{attribute 'linkalways'} 
{attribute 'no_explicit_call' := 'This FB is a CLASS and must be accessed using methods or properties'}
{attribute 'enable_dynamic_creation'}
FUNCTION_BLOCK _TIMESTRUCT EXTENDS StructuredDatatypeBase
VAR
	localData : TIMESTRUCT;
	activeData : REFERENCE TO TIMESTRUCT REF= localData;
	_wYear : _WORD(localData.wYear);
	_wMonth : _WORD(localData.wMonth);
END_VAR

PROPERTY PUBLIC Address : PVOID
GET
Address := ADR(activeData);
END_GET
END_PROPERTY

METHOD PUBLIC ClearReference
VAR_INPUT
END_VAR
activeData REF= localData;
END_METHOD

METHOD PUBLIC Clone : I_Datatype
VAR
    pClone : POINTER TO _TIMESTRUCT;
END_VAR
pClone := __NEW(_TIMESTRUCT());
pClone^.Value := Value;
Clone := pClone^;
END_METHOD

PROPERTY PUBLIC Identifier : T_MAXSTRING
GET
Identifier := 'TIMESTRUCT';
END_GET
END_PROPERTY

METHOD PROTECTED InitializeMembers
VAR_INPUT
	members : REFERENCE TO MembersHost;
END_VAR
_wYear.MakeReferenceTo(activeData.wYear);
members.AddMember('wYear',_wYear);

_wMonth.MakeReferenceTo(activeData.wMonth);
members.AddMember('wMonth',_wMonth);
END_METHOD

METHOD PUBLIC MakeReferenceTo
VAR_INPUT
	ReferenceTarget : TIMESTRUCT;
END_VAR
activeData REF= ReferenceTarget;
END_METHOD

PROPERTY PUBLIC Size : UDINT
GET
Size := SIZEOF(activeData);
END_GET
END_PROPERTY

METHOD TryMakeReferenceTo : BOOL
VAR_INPUT
	Target : I_Datatype;
END_VAR
VAR
	pTargetData : POINTER TO TIMESTRUCT;
END_VAR
IF NOT (Target.IecType = IecType) THEN
	RETURN;
END_IF

pTargetData := Target.Address;
activeData REF= pTargetData^;
TryMakeReferenceTo := TRUE;
END_METHOD

PROPERTY PUBLIC Value : TIMESTRUCT
GET
Value := activeData;
END_GET
SET
activeData := Value;
END_SET
END_PROPERTY

PROPERTY PUBLIC wMonth : Reference to _WORD
GET
wMonth := _wMonth;
END_GET
END_PROPERTY

PROPERTY PUBLIC wYear : Reference to _WORD
GET
wYear := _wYear;
END_GET
END_PROPERTY

END_FUNCTION_BLOCK

(* stored: Version 1.1.0.1, ProductVersion 3.1.4024.12
   POU _TIMESTRUCT: Id {82e9ef09-f63f-071f-12cd-f370d2802325}, SpecialFunc None
   Folder Protected: Id {9fdedf6e-4ca0-00e0-0273-13cb491dabf3}
   Property Address: Id {b5129746-2857-0022-1d98-5cd0054c1e32}
   Get Get: Id {b9ad7187-0100-02be-2dd1-43dd70cfdd46}
   Method ClearReference: Id {16c22b7d-2069-0e94-0823-7f69befe1715}
   Method Clone: Id {f9cc5498-2141-4519-8b72-11d757b9f1bd}
   Property Identifier: Id {11804f6c-c92e-0f5b-382d-3367d277dbcc}
   Get Get: Id {7977c071-5d37-04dd-33f0-5d682f8e3abf}
   Method InitializeMembers: Id {59fd7717-5550-0f25-158c-9c1e87cde269}
   Method MakeReferenceTo: Id {7e8e9cd2-b76b-014b-0b95-9790b062a9ee}
   Property Size: Id {3db85a58-3871-08be-0a1b-c8cbab28906e}
   Get Get: Id {c45ad51d-3dc4-00ea-11f7-a16d1bad1963}
   Method TryMakeReferenceTo: Id {8b5d5a6b-3b1b-05bb-2e0f-edb7929e5540}
   Property Value: Id {b58f9a32-1b3b-0a05-0577-0e7b74707ce6}
   Get Get: Id {d1a2ef74-1fb0-0703-20c2-eb9eec1cc598}
   Set Set: Id {4bd1c6bf-61b3-0a38-37ec-840667c35baf}
   Property wMonth: Id {54bb8911-1454-0b68-0e6e-66985ac5d437}
   Get Get: Id {8a1a1f3d-9a7a-02bf-2086-eb0b47f7f038}
   Property wYear: Id {3419be73-53a1-06fe-0591-dafdced19fef}
   Get Get: Id {aaabb8ed-77b5-04e0-2779-9412c3abbc56} *)
